Staubli VAL3: getNextSequenceNumber.pgx

program getNextSequenceNumber(num& x_nSequenceNumber)
begin
    x_nSequenceNumber = x_nSequenceNumber + 1
    if (x_nSequenceNumber > 65535)
      // Wrap around (uint16_t)
      x_nSequenceNumber = 0
    endIf

end
